// Mitsubishi GX Works2 project: bit_control_shift_rotate   PLC: Q02/Q02H

PROGRAM bitctrl
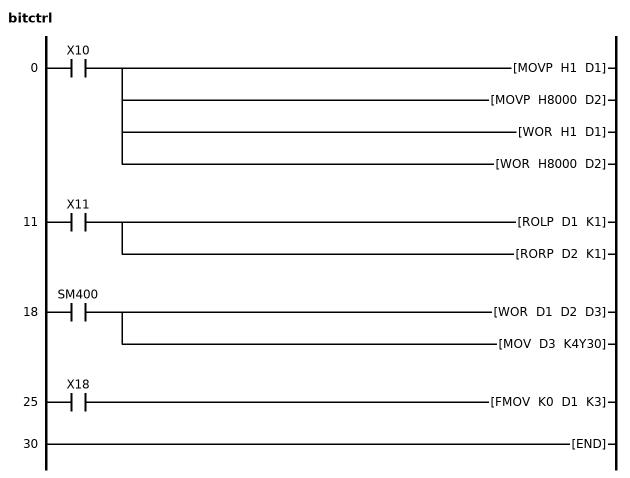
0     LD      X10
      MOVP    H1 D1
      MOVP    H8000 D2
      WOR     H1 D1
      WOR     H8000 D2
11    LD      X11
      ROLP    D1 K1
      RORP    D2 K1
18    LD      SM400
      WOR     D1 D2 D3
      MOV     D3 K4Y30
25    LD      X18
      FMOV    K0 D1 K3
30    END
END_PROGRAM

PROGRAM noENC
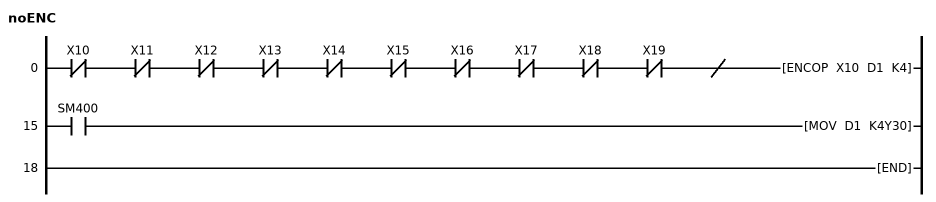
0     LDI     X10
      ANI     X11
      ANI     X12
      ANI     X13
      ANI     X14
      ANI     X15
      ANI     X16
      ANI     X17
      ANI     X18
      ANI     X19
      INV
      ENCOP   X10 D1 K4
15    LD      SM400
      MOV     D1 K4Y30
18    END
END_PROGRAM
